PROGRAM MAIN
VAR
	MCPower: MC_Power;
	McJog: MC_Jog;
	McReadStatus: MC_ReadStatus;
	McMoveVelocity: MC_MoveVelocity;
	McHalt: MC_Halt;
END_VAR

EnableAxis();
Jog();
MoveVelocity();
Halt();
ReadStatus();

ACTION EnableAxis:
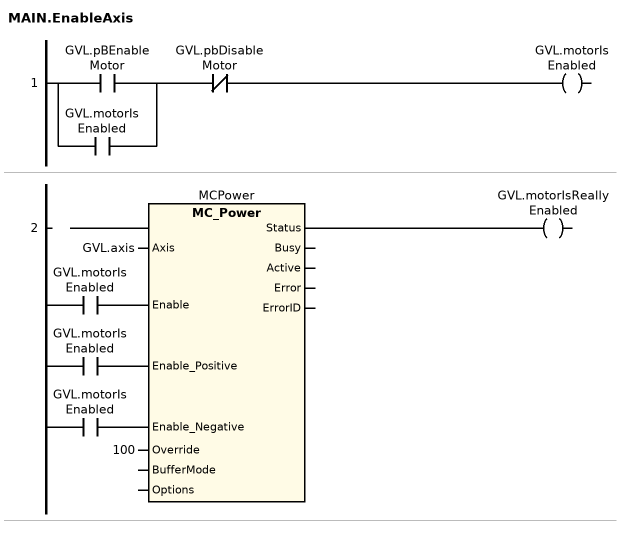
// NETWORK 1
GVL.motorIsEnabled := (GVL.pBEnableMotor OR GVL.motorIsEnabled) AND NOT GVL.pbDisableMotor;

// NETWORK 2
MCPower(
    Axis := GVL.axis,
    Enable := GVL.motorIsEnabled,
    Enable_Positive := GVL.motorIsEnabled,
    Enable_Negative := GVL.motorIsEnabled,
    Override := 100); // MC_Power
GVL.motorIsReallyEnabled := MCPower.Status;
END_ACTION

ACTION Halt:
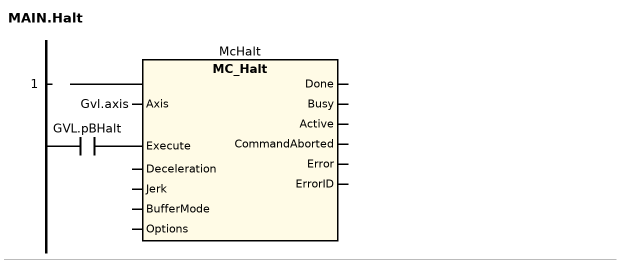
// NETWORK 1
McHalt(Axis := Gvl.axis, Execute := GVL.pBHalt); // MC_Halt
END_ACTION

ACTION Jog:
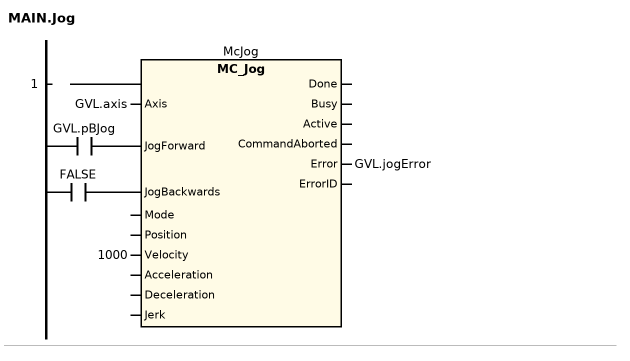
// NETWORK 1
McJog(
    Axis := GVL.axis,
    JogForward := GVL.pBJog,
    JogBackwards := FALSE,
    Velocity := 1000,
    Error => GVL.jogError); // MC_Jog
END_ACTION

ACTION MoveVelocity:
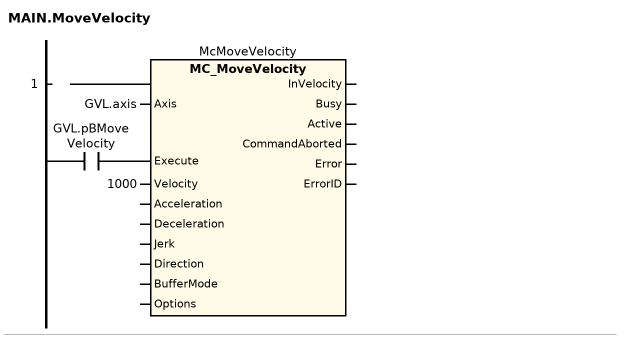
// NETWORK 1
McMoveVelocity(Axis := GVL.axis, Execute := GVL.pBMoveVelocity, Velocity := 1000); // MC_MoveVelocity
END_ACTION

ACTION ReadStatus:
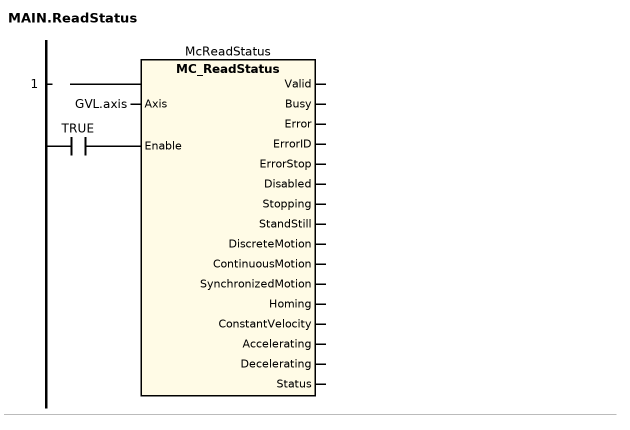
// NETWORK 1
McReadStatus(Axis := GVL.axis, Enable := TRUE); // MC_ReadStatus
END_ACTION

END_PROGRAM

(* stored: Version 1.1.0.1, ProductVersion 3.1.4024.12
   POU MAIN: Id {fd475419-3652-4af7-8ed4-30b0790529c7}, SpecialFunc None
   Action EnableAxis: Id {07a61e8a-3dba-4650-ad3b-ad452b06be21}
   Action Halt: Id {f8aed090-fa70-4d03-bc19-5abaf931d368}
   Action Jog: Id {64897d62-091a-4ac9-b417-db3c97dc6201}
   Action MoveVelocity: Id {2d778022-c8a6-4738-abb5-c6e7a6d72a39}
   Action ReadStatus: Id {fa75e5b9-7097-448d-a928-c15926b5fcac} *)
